// TIA Portal V19 export
FUNCTION_BLOCK "FB_FW_MANAGER"   // FB1, STL
{ S7_Optimized_Access := 'FALSE' }
AUTHOR : MS
// stored: AutoNumber false
   VAR_INPUT
      CallDBNr : DB_ANY;
   END_VAR
   VAR
      leng : Int := 18;
      Offset : Int := 50;
      resDW_1 : DWord;
      resDW_2 : DWord;
      resDW_3 : DWord;
      resDW_4 : DWord;
      Kettenpos : Array[1..4] of Byte;   // Positionen für Ketten (z.Bsp. Optimierungsergebnisse)
      Auto : Struct
         Anlage : Bool;
         Reihe_1 : Bool;
         Reihe_2 : Bool;
         Reihe_3 : Bool;
         Reihe_4 : Bool;
         Reihe_5 : Bool;
         res : Bool;
         res_1 : Bool;
         Anlage_not : Bool;
         Reihe_not_1 : Bool;
         Reihe_not_2 : Bool;
         Reihe_not_3 : Bool;
         Reihe_not_4 : Bool;
         Reihe_not_5 : Bool;
         res_2 : Bool;
         res_3 : Bool;
      END_STRUCT;
      resDW_6 : DWord;
      resDW_7 : DWord;
      resDW_8 : DWord;
      resDW_9 : DWord;
      resW : Int;
      akt_CT : Int;   // aktuelle SPS-Zykluszeit
      max_CT : Int;   // maximale SPS-Zykluszeit
      FW_DAT : Array[1..20] of Struct
         WT_NR_LANG : DInt;
         IST_POS : Byte;
         ZIEL_POS : Byte;
         Fahrt_Vor : Bool;
         Fahrt_Rck : Bool;
         Heben : Bool;
         Senken : Bool;
         Bereit : Bool;
         Fehler : Bool;
         Dummy : Bool;
         res : Bool;
         Tipp : Bool;
         Hand : Bool;
         Auto_Stop : Bool;
         Auto : Bool;
         Halt : Bool;
         K_Auto : Bool;
         Kette_wait_Start : Bool;
         Kette_wait_Ende : Bool;
         Unten : Bool;
         Z_Sensor : Bool;
         Oben : Bool;
         mittig : Bool;
         HWmittig : Bool;
         res_7 : Bool;
         res_8 : Bool;
         res_9 : Bool;
         WT_DB_Nr : Byte;
         IstInc : DInt;
         Stangen_Nr : Byte;
         WT_Typ : Byte;
         priorisirt : Bool;
         in_Anlage : Bool;
         in_Entmetall : Bool;
         aus_Anlage : Bool;
         aus_Entmetall : Bool;
         Speicherprog : Bool;
         Trommel : Bool;
         Leer_WT : Bool;
         BefX : Byte;
      END_STRUCT;
   END_VAR
   VAR_TEMP
      DB_Nr : Int;
      Kette_DB : Word;
      Count : Byte;
      TaktKette : Bool;
      Systime : Time;
   END_VAR
BEGIN

NETWORK
TITLE = 
//----------------------------------
//Initialisieren
//----------------------------------
      SET;
      R     #Auto.Anlage;
      R     #Auto.Reihe_1;
      R     #Auto.Anlage_not;
      R     #Auto.Reihe_not_1;

//----------------------------------
//Kommunikation zwischen FWs
      CALL  "FC_FW_Bereich";

//----------------------------------
//Rücksetzen der FW-Signale im Bad
      CALL  "FC_Reset_FWBits_im_Bad"
      ( Reset_in_out_nen := FALSE
      );


NETWORK
TITLE = Betriebsarten überprüfen
//----------------------------------
//Betriebsart-Check FW
//----------------------------------
      A     "DI_FW_1".ZST.Auto;
      S     #Auto.Anlage;
      S     #Auto.Reihe_1;
      NOT;
      S     #Auto.Anlage_not;
      S     #Auto.Reihe_not_1;


NETWORK
TITLE = FW-Bearbeitung
//----------------------------------
//FW Bearbeitung
//----------------------------------
      CALL  TIME_TCK
      ( RET_VAL := #Systime
      );

      L     #Systime;
      L     16#7FFF_FFFF;
      AD;
      T     #Systime;

      CALL  "FB_FW_x", "DI_FW_1";

//---------------------------
//FW-Bearbeitung Fahren
//---------------------------

      CALL  "FB_POS_FW_INC", "DI_FW_POS_1"
      ( SysTime := #Systime
      );

//---------------------------
//FW-Bearbeitung Heben
//---------------------------

      CALL  "FB_HUB_FW_li", "DI_FW_HUB_links"
      ( FW_DBNr := 11,
        SysTime := #Systime
      );

      CALL  "FB_HUB_FW_re", "DI_FW_HUB_rechts"
      ( FW_DBNr := 11,
        SysTime := #Systime
      );

      SET;
      R     "DI_FW_1".IN.Com_Reset;


      CALL  "FC_Reset_FWBits_im_Bad"
      ( Reset_in_out_nen := TRUE
      );

NETWORK
TITLE = FW-Schieben
//---------------------------
//Fahrwagen schieben
//---------------------------
      CALL  "FC_FW_SCHIEBEN";


NETWORK
TITLE = Querförderer
//---------------------------
//WR02 / WR03
//---------------------------
      CALL  "FB_QF", "DI_QF_WR02_03";


END_FUNCTION_BLOCK
